{attribute 'linkalways'} 
{attribute 'no_explicit_call' := 'This FB is a CLASS and must be accessed using methods or properties'}
{attribute 'enable_dynamic_creation'}
FUNCTION_BLOCK Node_F_VN_LaplacianFilter EXTENDS Node
VAR
	ipSrcImage : _ITcVnImage;
    ipDestImage : _ITcVnImage;
    eDestDepth : _ETcVnElementType(ETcVnElementType.TCVN_ET_SAME_AS_SOURCE);
    hrPrev : _HRESULT(S_OK);
	hresult : _HRESULT(S_OK);
END_VAR

METHOD PUBLIC  Clone : I_Node
VAR
	pNode : POINTER TO Node_F_VN_LaplacianFilter;
END_VAR
pNode := __NEW(Node_F_VN_LaplacianFilter);
Clone := pNode^;
END_METHOD

METHOD FB_init : BOOL
VAR_INPUT
	bInitRetains : BOOL; // if TRUE, the retain variables are initialized (warm start / cold start)
	bInCopyCode : BOOL;  // if TRUE, the instance afterwards gets moved into the copy code (online change)
END_VAR
AddInput('ipSrcImage', ipSrcImage);
AddInput('hrPrev', hrPrev);
AddOutput('ipDestImage', ipDestImage);
AddOutput('hresult',hresult);
AddParameter('eDestDepth', eDestDepth);
END_METHOD

METHOD PROTECTED  OnExecute : HRESULT
hresult.Value := F_VN_LaplacianFilter(
	ipSrcImage := ipSrcImage.Value, 
	ipDestImage := ipDestImage.Value, 
	eDestDepth := eDestDepth.Value, 
	hrPrev := hrPrev.Value);
END_METHOD

END_FUNCTION_BLOCK

(* stored: Version 1.1.0.1, ProductVersion 3.1.4024.13
   POU Node_F_VN_LaplacianFilter: Id {69e65283-ace7-0c55-30fa-949b5a402b03}, SpecialFunc None
   Folder Constructor: Id {3683372b-8bce-09b7-2df1-f23e93a3b6fa}
   Method Clone: Id {7cc768b2-50e5-0afc-3b0f-89165a9d0e71}
   Method FB_init: Id {3353b323-7152-0b56-272d-6c7bb3991130}
   Method OnExecute: Id {0e14aa31-08be-0513-0ab6-f2d326d3028a} *)
